(* CODESYS project praca.ecp

Project tree, tasks and I/O mapping:
  PFC200_2ETH_RS : 750-8202 PFC200 2ETH RS, WAGO, order no. 0750-8202, version 5.14.3.63
    application Application
      libraries: ; WagoAppControlSuite, 1.0.1.4 (WAGO); Util, * (System)
      task PLC_Task (cyclic, interval t#50ms, priority 15) calls Main
      program PLC_PRG [ST]
      program POU_1 [LD]
      program POU [LD]
      program Main [ST]
    Kbus : Kbus, WAGO, version 1.4.0.2
        unmapped channels: K-BUS diagnostics
      _2_DO_Generic : 075x-2DO, WAGO, order no. 075x-2DO, version 0.0.0.13
          settings: K-BUS Module slot index = 1
          output Application.PLC_PRG.went_on : BOOL  // _OUT._OUT
          unmapped channels: _OUT
      _4AI_0_10_VDC_SE : 0750-0459, WAGO, order no. 0750-0459, version 0.0.0.13
          settings: K-BUS Module slot index = 2
          input  Application.PLC_PRG.pomiar_temp : WORD  // _IW 1
          unmapped channels: _IW 2, _IW 3, _IW 4
      _4AO_4_20mA : 0750-0555, WAGO, order no. 0750-0555, version 0.0.0.12
          settings: K-BUS Module slot index = 3
          output Application.PLC_PRG.grzaka_ster : WORD  // _QW 1
          unmapped channels: _QW 2, _QW 3, _QW 4
    MODBUS
      MODBUS : MODBUS, WAGO, order no. n/a, version 1.1.1.15
        LocalDeviceModbus : MODBUS Slave, WAGO, order no. n/a, version 1.1.1.15
          TcpSettings : Modbus TCP Slave, WAGO, order no. n/a, version 1.1.1.15
              settings: TCP connection watchdog = 200 10ms
    Serial
      COM1 : COM1, WAGO, version 0.0.0.19
  Generic_Modbus_Master : ThirdParty Modbus Master, WAGO, order no. GenericModbusMaster, version 1.0.0.1
*)

// PFC200_2ETH_RS/Application/Main
PROGRAM Main
VAR
END_VAR

//PLC_PRG();
//POU();
POU_1();

END_PROGRAM

// PFC200_2ETH_RS/Application/PLC_PRG
PROGRAM PLC_PRG
VAR
	went_on:BOOL;
	
	pomiar_temp: int;
	
	grzaka_ster: INT;
	
END_VAR

IF pomiar_temp>0 THEN
	went_on:=TRUE;
	
ELSE
	went_on:=FALSE;
END_IF

END_PROGRAM

// PFC200_2ETH_RS/Application/POU
PROGRAM POU
VAR
	FbTemperatureControlContinous_01_0: WagoAppControlSuite.FbTemperatureControlContinous_01;
	en_pid AT %MB100: BOOL;
	tmp_zadana: REAL;
	probkowanie: TIME := T#1s;
	en_ext_control_param: BOOL;
	rKp: REAL;
	rTn: REAL;
	rTv: REAL;
	rOmax: REAL := 0.0;
	rOmin: REAL := 32767.0;
	en_man_op: BOOL;
	rManVal: REAL;
	stryctConf: typTempConfiguration_01;
	en_rel_by_op: BOOL;
	rStatVal: REAL;
	en_dis_pt1: BOOL;
	enAutoTune: BOOL;
	reset_pid: BOOL;
	wysterowanie: REAL;
	rKs: REAL;
	rTu: REAL;
	rTg: REAL;
	problem: BOOL;
	xLimReached: BOOL;
	xLimMaxReached: BOOL;
	xLimMinReached: BOOL;
	iStatus: INT;
	sStatus: STRING;
	actKp: REAL;
	actTn: REAL;
	actTv: REAL;
END_VAR

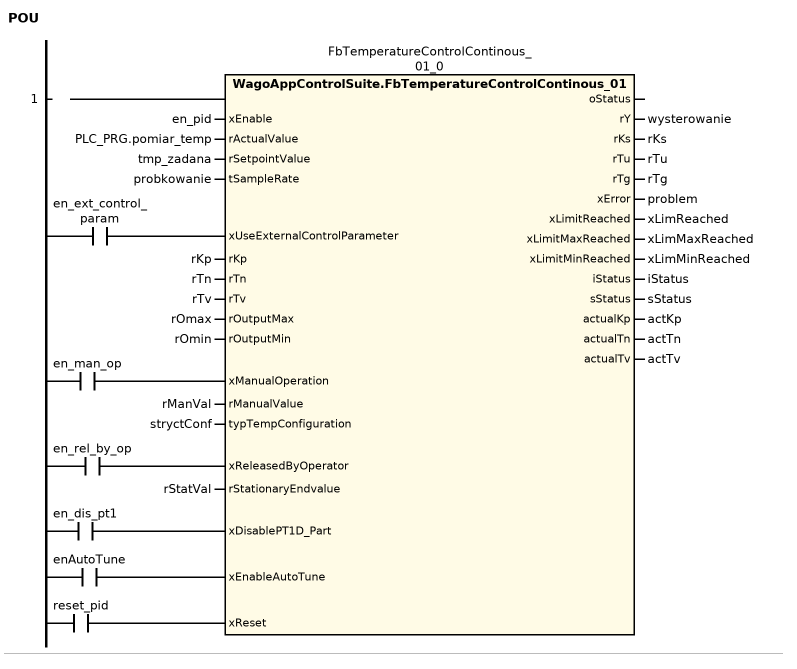
// NETWORK 1
FbTemperatureControlContinous_01_0(
    xEnable := en_pid,
    rActualValue := PLC_PRG.pomiar_temp,
    rSetpointValue := tmp_zadana,
    tSampleRate := probkowanie,
    xUseExternalControlParameter := en_ext_control_param,
    rKp := rKp,
    rTn := rTn,
    rTv := rTv,
    rOutputMax := rOmax,
    rOutputMin := rOmin,
    xManualOperation := en_man_op,
    rManualValue := rManVal,
    typTempConfiguration := stryctConf,
    xReleasedByOperator := en_rel_by_op,
    rStationaryEndvalue := rStatVal,
    xDisablePT1D_Part := en_dis_pt1,
    xEnableAutoTune := enAutoTune,
    xReset := reset_pid,
    rY => wysterowanie,
    rKs => rKs,
    rTu => rTu,
    rTg => rTg,
    xError => problem,
    xLimitReached => xLimReached,
    xLimitMaxReached => xLimMaxReached,
    xLimitMinReached => xLimMinReached,
    iStatus => iStatus,
    sStatus => sStatus,
    actualKp => actKp,
    actualTn => actTn,
    actualTv => actTv); // WagoAppControlSuite.FbTemperatureControlContinous_01

END_PROGRAM

// PFC200_2ETH_RS/Application/POU_1
PROGRAM POU_1
VAR
	PID_0: Util.PID;
	en_simple_man: BOOL;
	en_reset_man: BOOL;
	lim_act: BOOL;
	overflow: BOOL;
	act_val: REAL;
	set_pt: REAL;
	kp: REAL;
	tn: REAL;
	tv: REAL;
	y_man: REAL;
	y_offset: REAL;
	y_min: REAL;
	y_max: REAL;
END_VAR

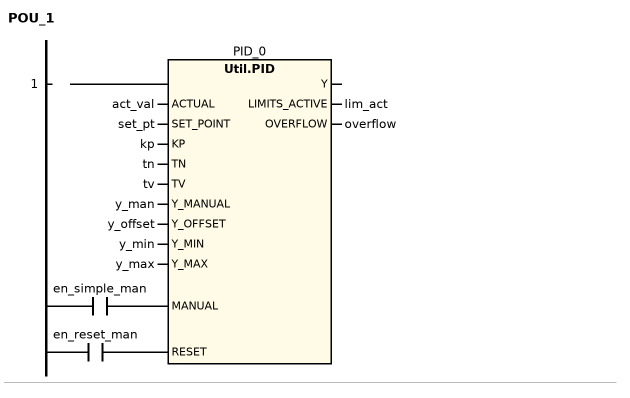
// NETWORK 1
PID_0(
    ACTUAL := act_val,
    SET_POINT := set_pt,
    KP := kp,
    TN := tn,
    TV := tv,
    Y_MANUAL := y_man,
    Y_OFFSET := y_offset,
    Y_MIN := y_min,
    Y_MAX := y_max,
    MANUAL := en_simple_man,
    RESET := en_reset_man,
    LIMITS_ACTIVE => lim_act,
    OVERFLOW => overflow); // Util.PID

END_PROGRAM
